// TIA Portal V19 export
TYPE "lexchangetray_typeroller_signalTM_Cmd_1"
// Type: Bool
// stored: Access Published
   STRUCT
      simActive : Bool;
   END_STRUCT;
END_TYPE
